PROGRAM MAIN
VAR
END_VAR


//PRG_CSVRead();
//PRG_CSVWrite();

//Call Programs
PRG_Simulator();
PRG_ReadTime();

END_PROGRAM

(* stored: Version 1.1.0.1, ProductVersion 3.1.4024.12
   POU MAIN: Id {4d940c54-4155-4073-8351-63edeb64b412}, SpecialFunc None *)
